# EPICS autosave request: ioc/AutoSaveRestore/rampSetting.req
$(P)$(R)VRAMPstepSize
$(P)$(R)VRAMPinterval
$(P)$(R)desiredHV
